TYPE ST_HMIConfiguration :
STRUCT
	ComponentConfiguration : REFERENCE TO ST_CommandConfiguration;
END_STRUCT
END_TYPE

(* stored: Version 1.1.0.1
   DUT ST_HMIConfiguration: Id {28fdd680-6f2c-4bae-96ec-4423cbed4ce3} *)
